// Mitsubishi GX Works2 project: group20 - final   PLC: FX3G

// global labels: Global1
VAR_GLOBAL
  startDay AT X007 : BOOL;
  raspberryInput AT D1112 : REAL;
  zero AT E0 : REAL;
  lemonInput AT D1115 : REAL;
  gumyBearsInput AT D1118 : REAL;
  outOfStock AT M1 : BOOL;
  emergencyButton AT X005 : BOOL;
  outOfStockHold AT M2 : BOOL;
  stablilizerInput AT D1121 : REAL;
  raspberryQuantity AT D1114 : REAL;
  lemonQuantity AT D1117 : REAL;
  gumyBearsQuantity AT D1120 : REAL;
  stabilizerQuantity AT D1123 : REAL;
  IC_regular AT M4 : BOOL;
  IC_special AT M5 : BOOL;
  Sample AT X001 : BOOL;
  analog_input_1 AT D8280 : INT;
END_VAR
VAR_GLOBAL CONSTANT
  normalization : REAL := 400;
END_VAR
VAR_GLOBAL
  Input_1 AT D1125 : REAL;
  IC_raspberry AT D1127 : REAL;
  IC_lemon AT D1129 : REAL;
END_VAR
VAR_GLOBAL CONSTANT
  cons_350 : REAL := 350;
  cons_490 : REAL := 490;
  cons_560 : REAL := 560;
  cons_700 : REAL := 700;
  cons_280 : REAL := 280;
  cons_455 : REAL := 455;
  cons_105 : REAL := 105;
  cons_385 : REAL := 385;
  cons_665 : REAL := 665;
  cons_210 : REAL := 210;
  timer_5_sec : INT := 50;
END_VAR
VAR_GLOBAL
  Y_0 AT Y000 : BOOL;
  TC_0 AT TC0 : BOOL;
END_VAR
VAR_GLOBAL CONSTANT
  min_raspberry : REAL := 280;
  min_lemon : REAL := 420;
  min_gumyBears : REAL := 28;
END_VAR
VAR_GLOBAL
  Y_7 AT Y007 : BOOL;
  endDay AT M6 : BOOL;
  TS_0 AT TS0 : BOOL;
END_VAR
VAR_GLOBAL CONSTANT
  regular_group : REAL := 5;
  special_group : REAL := 6;
END_VAR
VAR_GLOBAL
  endPerp AT M7 : BOOL;
  X_2 AT X002 : BOOL;
  fridge_raspberry AT D1131 : REAL;
  fridge_lemon AT D1133 : REAL;
  moved_to_fridge AT M8 : BOOL;
  TC_1 AT TC1 : BOOL;
END_VAR
VAR_GLOBAL CONSTANT
  timer_8_sec : INT := 80;
END_VAR
VAR_GLOBAL
  TS_1 AT TS1 : BOOL;
  X_3 AT X003 : BOOL;
  Y_2 AT Y002 : BOOL;
  mix_container AT D1135 : REAL;
  gumyBears_mix AT D1137 : REAL;
END_VAR
VAR_GLOBAL CONSTANT
  cons_28 : REAL := 28;
  cons_70 : REAL := 70;
  cons_3 : REAL := 3;
END_VAR
VAR_GLOBAL
  mix_time AT D1139 : REAL;
END_VAR
VAR_GLOBAL CONSTANT
  cons_5 : REAL := 5;
END_VAR
VAR_GLOBAL
  end_fridge AT M9 : BOOL;
  monitoring_lighter AT M10 : BOOL;
  startBlink AT M11 : BOOL;
END_VAR
VAR_GLOBAL CONSTANT
  timer_3_sec : INT := 30;
END_VAR
VAR_GLOBAL
  TS_2 AT TS2 : BOOL;
  stop_blink_after AT M12 : BOOL;
  timerBlink1 AT TC3 : BOOL;
  timerBlink2 AT TC4 : BOOL;
  mixTimer AT TC2 : BOOL;
END_VAR
VAR_GLOBAL CONSTANT
  timeBlink1 : INT := 10;
  timeBlink2 : INT := 10;
END_VAR
VAR_GLOBAL
  end_timeBlink1 AT TS3 : BOOL;
  end_timeBlink2 AT TS4 : BOOL;
  Y_5 AT Y005 : BOOL;
  Y_6 AT Y006 : BOOL;
  X_4 AT X004 : BOOL;
  mixTimer1 AT TC5 : BOOL;
  TS_5 AT TS5 : BOOL;
END_VAR
VAR_GLOBAL CONSTANT
  package_7 : INT := 7;
END_VAR
VAR_GLOBAL
  Y_4 AT Y004 : BOOL;
  start_packing AT M13 : BOOL;
  X_0 AT X000 : BOOL;
  package_container AT D1141 : REAL;
END_VAR
VAR_GLOBAL CONSTANT
  cons_1 : REAL := 1;
END_VAR
VAR_GLOBAL
  output AT D1143 : REAL;
  analog_output AT D8282 : INT;
  stop_y4 AT M14 : BOOL;
  package_counter AT CC2 : BOOL;
  CS_2 AT CS2 : BOOL;
  stop_m4 AT M15 : BOOL;
END_VAR
VAR_GLOBAL CONSTANT
  normalization_2 : REAL := 40;
END_VAR

// task Task_01 (event TRUE, interval 0, priority 31): POU_01

PROGRAM POU_01
(* structured ladder/FBD written out as ST: instructions are called as NAME(EN, inputs, outputs); _pN, _eN, _tN stand for wires *)
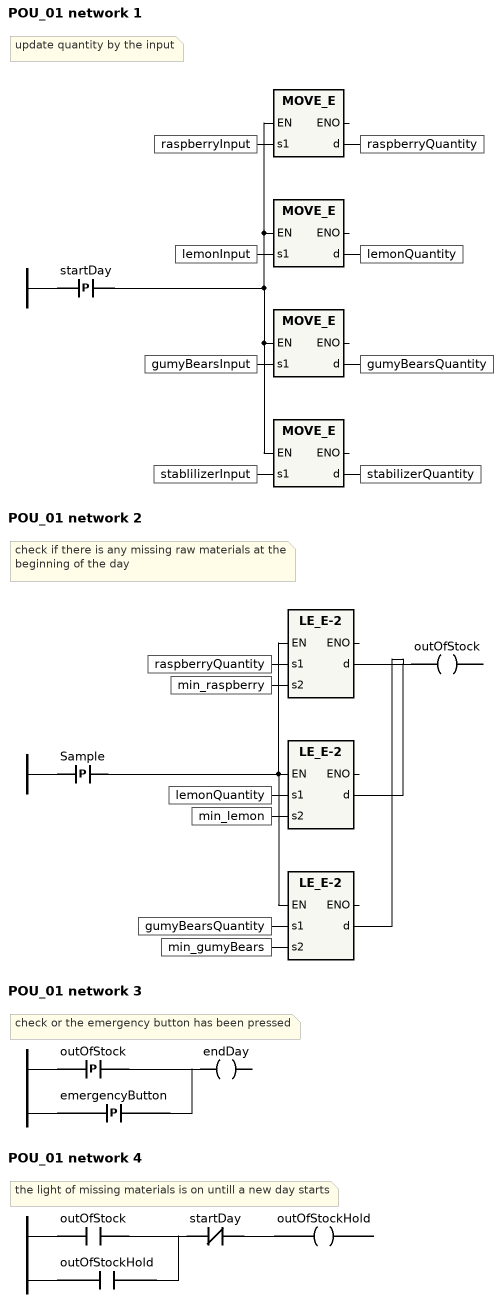
(* network 1 *)
(* update quantity by the input *)
_p1 := LDP(TRUE, startDay);
MOVE_E(_p1, raspberryInput, raspberryQuantity);
MOVE_E(_p1, lemonInput, lemonQuantity);
MOVE_E(_p1, gumyBearsInput, gumyBearsQuantity);
MOVE_E(_p1, stablilizerInput, stabilizerQuantity);
(* network 2 *)
(* check if there is any missing raw materials at the beginning of the day *)
_p1 := LDP(TRUE, Sample);
LE_E(_p1, raspberryQuantity, min_raspberry, _t2);
LE_E(_p1, lemonQuantity, min_lemon, _t3);
LE_E(_p1, gumyBearsQuantity, min_gumyBears, _t4);
outOfStock := _t2 OR _t3 OR _t4;
(* network 3 *)
(* check or the emergency button has been pressed *)
endDay := LDP(TRUE, outOfStock) OR LDP(TRUE, emergencyButton);
(* network 4 *)
(* the light of missing materials is on untill a new day starts *)
outOfStockHold := (outOfStock OR outOfStockHold) AND NOT startDay;
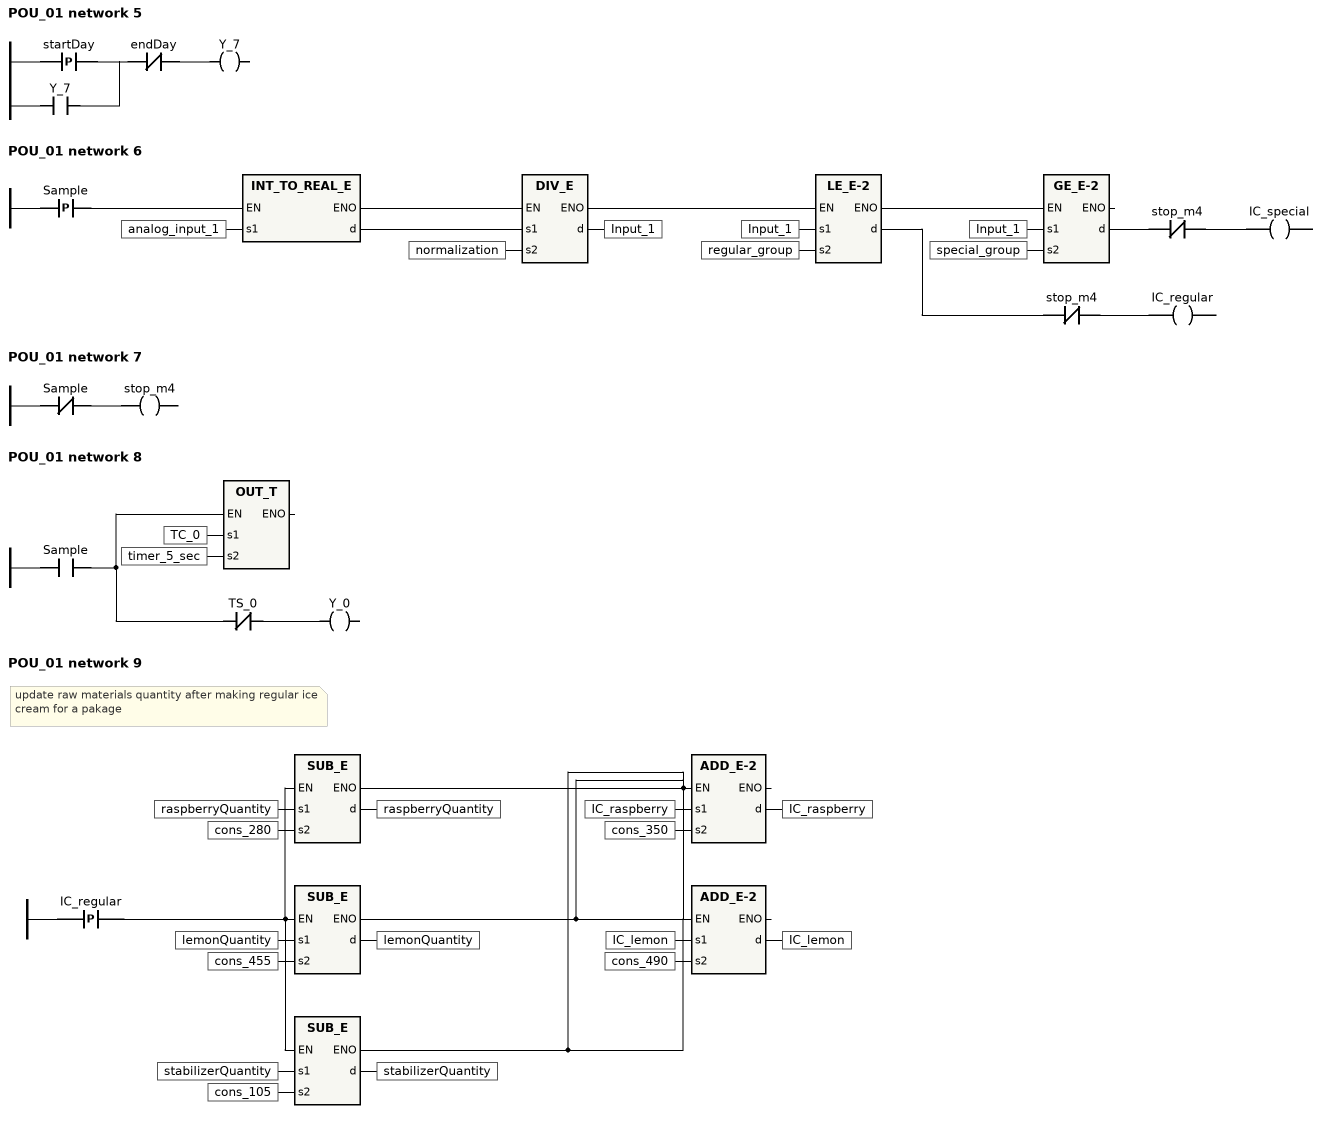
(* network 5 *)
Y_7 := (LDP(TRUE, startDay) OR Y_7) AND NOT endDay;
(* network 6 *)
_e2 := INT_TO_REAL_E(LDP(TRUE, Sample), analog_input_1, _t1);
_e3 := DIV_E(_e2, _t1, normalization, Input_1);
_e5 := LE_E(_e3, Input_1, regular_group, _t4);
GE_E(_e5, Input_1, special_group, _t6);
IC_special := _t6 AND NOT stop_m4;
IC_regular := _t4 AND NOT stop_m4;
(* network 7 *)
stop_m4 := NOT Sample;
(* network 8 *)
OUT_T(Sample, TC_0, timer_5_sec);
Y_0 := Sample AND NOT TS_0;
(* network 9 *)
(* update raw materials quantity after making regular ice cream for a pakage *)
_p1 := LDP(TRUE, IC_regular);
_e2 := SUB_E(_p1, raspberryQuantity, cons_280, raspberryQuantity);
_e3 := SUB_E(_p1, lemonQuantity, cons_455, lemonQuantity);
_e4 := SUB_E(_p1, stabilizerQuantity, cons_105, stabilizerQuantity);
_p5 := _e2 OR _e3 OR _e4;
ADD_E(_p5, IC_raspberry, cons_350, IC_raspberry);
ADD_E(_p5, IC_lemon, cons_490, IC_lemon);
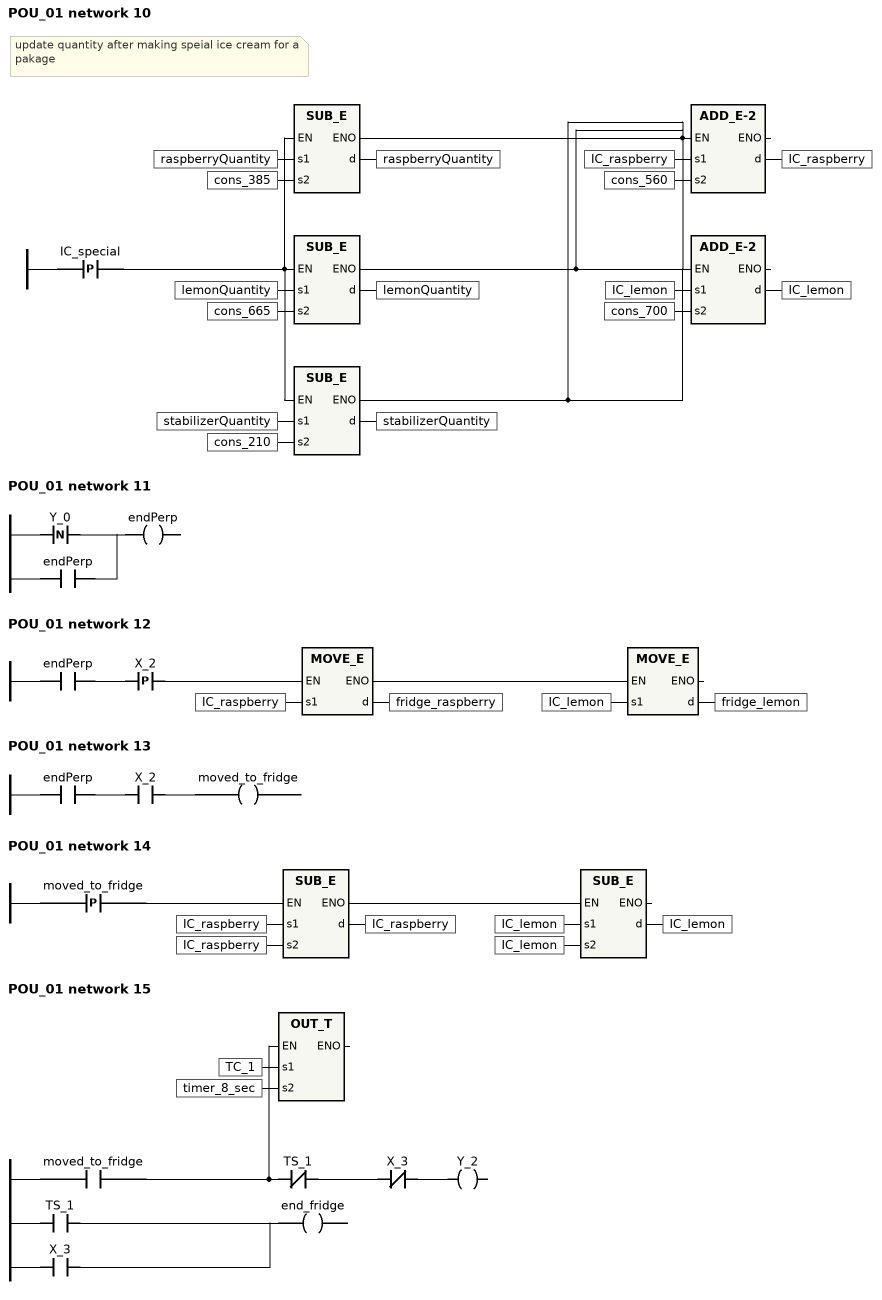
(* network 10 *)
(* update quantity after making speial ice cream for a pakage *)
_p1 := LDP(TRUE, IC_special);
_e2 := SUB_E(_p1, raspberryQuantity, cons_385, raspberryQuantity);
_e3 := SUB_E(_p1, lemonQuantity, cons_665, lemonQuantity);
_e4 := SUB_E(_p1, stabilizerQuantity, cons_210, stabilizerQuantity);
_p5 := _e2 OR _e3 OR _e4;
ADD_E(_p5, IC_raspberry, cons_560, IC_raspberry);
ADD_E(_p5, IC_lemon, cons_700, IC_lemon);
(* network 11 *)
endPerp := LDF(TRUE, Y_0) OR endPerp;
(* network 12 *)
_e1 := MOVE_E(endPerp AND LDP(TRUE, X_2), IC_raspberry, fridge_raspberry);
MOVE_E(_e1, IC_lemon, fridge_lemon);
(* network 13 *)
moved_to_fridge := endPerp AND X_2;
(* network 14 *)
_e1 := SUB_E(LDP(TRUE, moved_to_fridge), IC_raspberry, IC_raspberry, IC_raspberry);
SUB_E(_e1, IC_lemon, IC_lemon, IC_lemon);
(* network 15 *)
OUT_T(moved_to_fridge, TC_1, timer_8_sec);
Y_2 := moved_to_fridge AND NOT TS_1 AND NOT X_3;
end_fridge := TS_1 OR X_3;
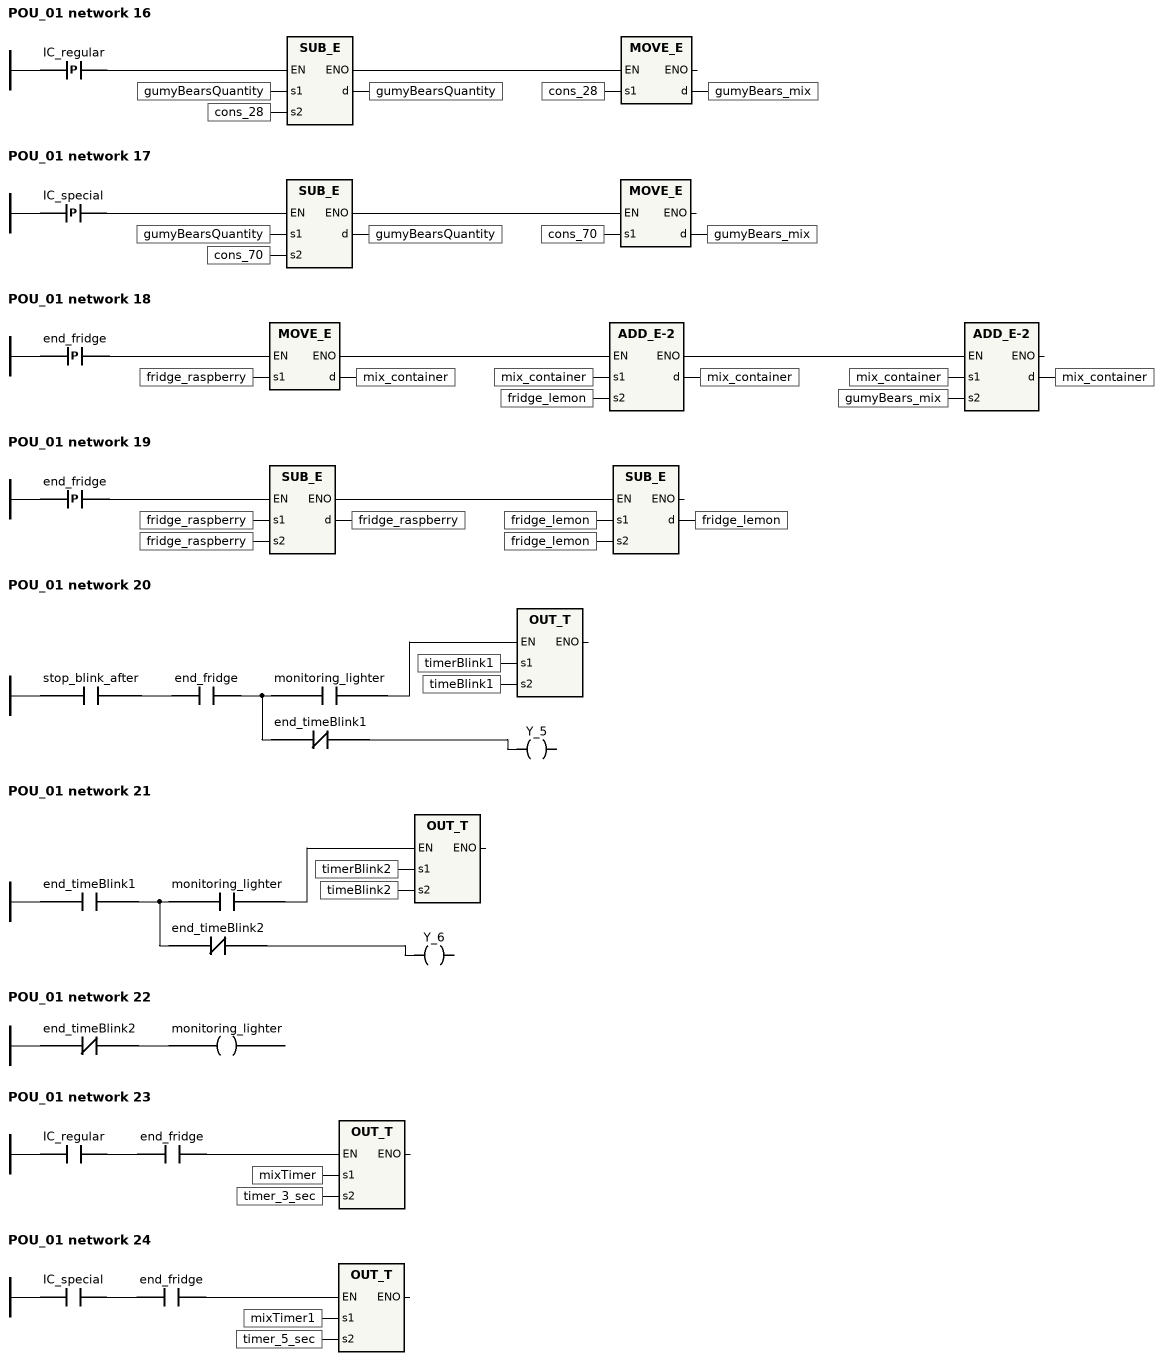
(* network 16 *)
_e1 := SUB_E(LDP(TRUE, IC_regular), gumyBearsQuantity, cons_28, gumyBearsQuantity);
MOVE_E(_e1, cons_28, gumyBears_mix);
(* network 17 *)
_e1 := SUB_E(LDP(TRUE, IC_special), gumyBearsQuantity, cons_70, gumyBearsQuantity);
MOVE_E(_e1, cons_70, gumyBears_mix);
(* network 18 *)
_e1 := MOVE_E(LDP(TRUE, end_fridge), fridge_raspberry, mix_container);
_e2 := ADD_E(_e1, mix_container, fridge_lemon, mix_container);
ADD_E(_e2, mix_container, gumyBears_mix, mix_container);
(* network 19 *)
_e1 := SUB_E(LDP(TRUE, end_fridge), fridge_raspberry, fridge_raspberry, fridge_raspberry);
SUB_E(_e1, fridge_lemon, fridge_lemon, fridge_lemon);
(* network 20 *)
_p1 := stop_blink_after AND end_fridge;
OUT_T(_p1 AND monitoring_lighter, timerBlink1, timeBlink1);
Y_5 := _p1 AND NOT end_timeBlink1;
(* network 21 *)
OUT_T(end_timeBlink1 AND monitoring_lighter, timerBlink2, timeBlink2);
Y_6 := end_timeBlink1 AND NOT end_timeBlink2;
(* network 22 *)
monitoring_lighter := NOT end_timeBlink2;
(* network 23 *)
OUT_T(IC_regular AND end_fridge, mixTimer, timer_3_sec);
(* network 24 *)
OUT_T(IC_special AND end_fridge, mixTimer1, timer_5_sec);
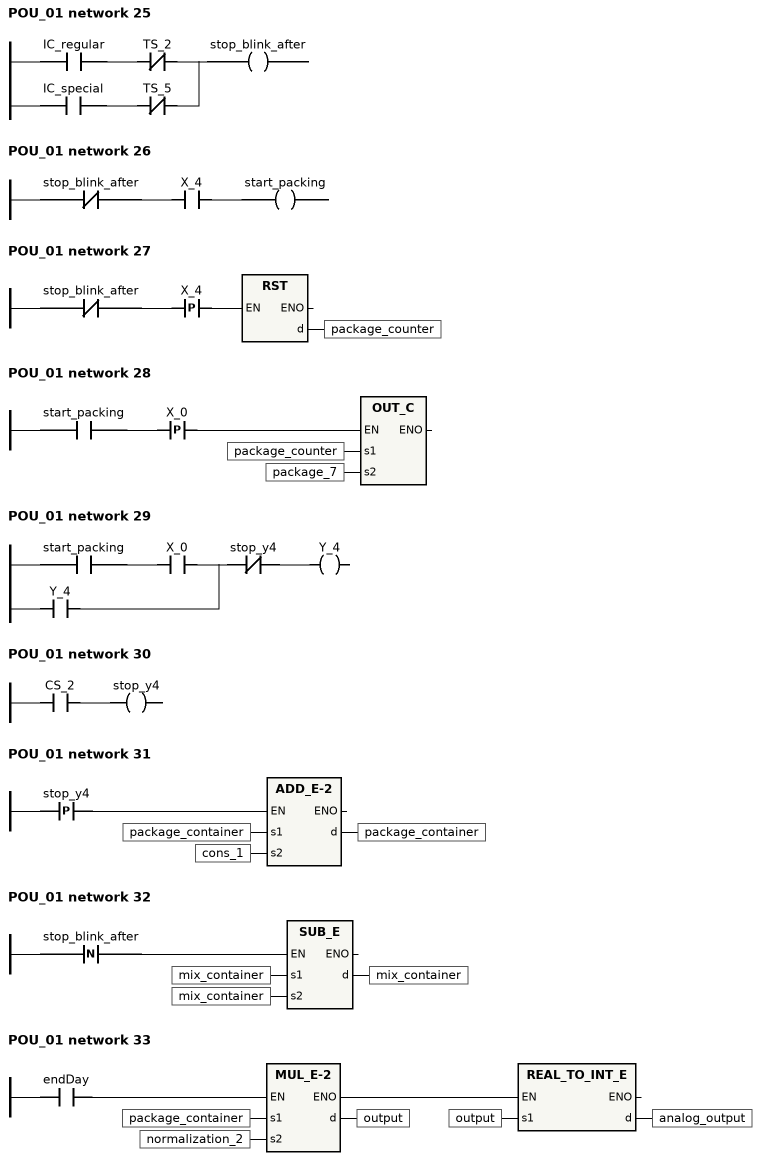
(* network 25 *)
stop_blink_after := (IC_regular AND NOT TS_2) OR (IC_special AND NOT TS_5);
(* network 26 *)
start_packing := NOT stop_blink_after AND X_4;
(* network 27 *)
RST(NOT stop_blink_after AND LDP(TRUE, X_4), package_counter);
(* network 28 *)
OUT_C(start_packing AND LDP(TRUE, X_0), package_counter, package_7);
(* network 29 *)
Y_4 := ((start_packing AND X_0) OR Y_4) AND NOT stop_y4;
(* network 30 *)
stop_y4 := CS_2;
(* network 31 *)
ADD_E(LDP(TRUE, stop_y4), package_container, cons_1, package_container);
(* network 32 *)
SUB_E(LDF(TRUE, stop_blink_after), mix_container, mix_container, mix_container);
(* network 33 *)
_e1 := MUL_E(endDay, package_container, normalization_2, output);
REAL_TO_INT_E(_e1, output, analog_output);
END_PROGRAM
